{attribute 'linkalways'}
{attribute 'no_explicit_call' := 'do not call this POU directly'}
FUNCTION_BLOCK InstanceCollection
VAR
	instances : ARRAY [0..MobjectCoreConstants.MAX_INSTANCES] OF I_Instance;
	last : DINT := EMPTY;
END_VAR
VAR CONSTANT
	EMPTY : DINT := -1;
END_VAR

PROPERTY PUBLIC Count : DINT
GET
Count := last + 1;
END_GET
END_PROPERTY

METHOD PUBLIC GetByIndex : I_Instance
VAR_INPUT
	Index : DINT;
END_VAR
GetByIndex := instances[Index];
END_METHOD

METHOD PUBLIC Insert
VAR_INPUT
	Instance : I_Instance;
END_VAR
last := last + 1;
instances[last] := Instance;
END_METHOD

METHOD Remove : BOOL
VAR_INPUT
	Instance : I_Instance;
END_VAR
VAR
	i: DINT;
END_VAR
FOR i := 0 TO last DO
	IF Instance = instances[i] THEN
		instances[i] := 0;
		
		IF i <> last THEN
			instances[i] := instances[last];
		END_IF
		
		last := last -1;
		
	END_IF
END_FOR
END_METHOD

END_FUNCTION_BLOCK

(* stored: Version 1.1.0.1, ProductVersion 3.1.4024.11
   POU InstanceCollection: Id {fa184060-a42a-4ff0-90e2-dcb283ec6dd8}, SpecialFunc None
   Property Count: Id {937cecfd-4306-400e-b623-8ba2f897672a}
   Get Get: Id {8e72a050-d6fe-4a19-a736-fd6abd2ef4e0}
   Method GetByIndex: Id {38bd5a7e-f9d7-4ee7-81f7-3b40a70ef39d}
   Method Insert: Id {12da7243-1afb-41ea-908d-6d963cadcc63}
   Method Remove: Id {5467eb59-5caf-4ef0-8c34-8e4adec7cb97} *)
